# EPICS substitutions: siteApps/EtherCat/m-epics-ecat2db/db/ecat2ek1101.substitutions
file ecat2ekxxxxID.template
{
	pattern {NULL}
		{NULL}

}

file ecat2slave.template
{
	pattern {DEVICENAME}
		{EK1101}
}
